// TwinCAT 3 PLC project Graham_PLC
// ProgramVersion: 3.1.4024.0
// libraries:
//   Tc2_Standard, * (Beckhoff Automation GmbH)
//   Tc2_System, * (Beckhoff Automation GmbH)
//   Tc3_Module, * (Beckhoff Automation GmbH)
// project tree:
//   GVLs/ GVL_HMI.TcGVL
//   / PlcTask.TcTTO
//   POUs/ MAIN.TcPOU, Signal_Generator.TcPOU
// real-time tasks:
//   TASK PlcTask: cycle T#10ms, priority 20, ADS port 350

CONFIGURATION Graham_PLC
    RESOURCE PLC ON TwinCAT3
        TASK PlcTask(INTERVAL := T#10ms, PRIORITY := 20);
        PROGRAM MAIN WITH PlcTask : MAIN;
    END_RESOURCE
END_CONFIGURATION

// ---- GVLs/GVL_HMI.TcGVL
{attribute 'qualified_only'}
VAR_GLOBAL
	lr_Heater1: LREAL;
	lr_Heater2: LREAL;
	lr_Heater3: LREAL;
END_VAR

// ---- POUs/MAIN.TcPOU
PROGRAM MAIN
VAR
END_VAR

Signal_Generator();

END_PROGRAM

// ---- POUs/Signal_Generator.TcPOU
PROGRAM Signal_Generator
VAR
	lr_Counter1: LREAL;
	lr_Counter2: LREAL;
	lr_Counter3: LREAL;
END_VAR

lr_Counter1:= lr_Counter1+0.005;
GVL_HMI.lr_Heater1:= SIN(lr_Counter1+3)*125+185;


lr_Counter2:= lr_Counter2+0.006;
GVL_HMI.lr_Heater2:= SIN(lr_Counter2)*120+180;

lr_Counter3:= lr_Counter3+0.008;
GVL_HMI.lr_Heater3:= COS(lr_Counter3)*130+190;

END_PROGRAM
